INTERFACE ITF_Clone

METHOD Clone : ITF_Cloneable
VAR_INPUT
END_VAR
END_METHOD

END_INTERFACE

(* stored: Version 1.1.0.1, ProductVersion 3.1.4024.12
   Itf ITF_Clone: Id {e61a57fe-4e8a-4d90-95ef-46051e43beee}
   Method Clone: Id {c3ef475b-c348-431b-881c-5199508ebca8} *)
